INTERFACE I_Syntax_Extended EXTENDS I_Syntax_Widget

METHOD M_Execute : BOOL
VAR_INPUT
    nCommand : DINT;
END_VAR
END_METHOD

METHOD M_Reset : BOOL
END_METHOD

PROPERTY P_ExtendedStatus : INT
GET
END_GET
END_PROPERTY

END_INTERFACE

(* stored: Version 1.1.0.1, ProductVersion 3.1.4024.16
   Itf I_Syntax_Extended: Id {13b41300-9ce0-4ce0-a29d-ee2f15951d9e}
   Method M_Execute: Id {e5f6a1b2-c3d4-4e5f-c06b-7c8d9e0f1a2b}
   Method M_Reset: Id {7ad8b0bd-b8e8-447e-ae70-6aaa2d45d1cc}
   Property P_ExtendedStatus: Id {acb160f8-190f-4161-806f-16a237f4e6af}
   Get Get: Id {5e573bf0-7431-42eb-99fa-2e7219b3fa95} *)
